TYPE ST_SafetyFunctionIn :
STRUCT
    byRaw : BYTE;
END_STRUCT
END_TYPE

(* stored: Version 1.1.0.1
   DUT ST_SafetyFunctionIn: Id {8070dc95-c87f-07f6-3fb8-b169434ba19a} *)
